FUNCTION_BLOCK PMLStateMachine IMPLEMENTS IPmlStateMachine
VAR_INPUT
END_VAR
VAR_OUTPUT
END_VAR
VAR
	_pmlStateMachine : Tc3_PackML_V2.PML_StateMachine;
	
END_VAR

_pmlStateMachine();

METHOD PUBLIC getState : E_PMLState
VAR_INPUT
END_VAR
getState := _pmlStateMachine.eState;
END_METHOD

METHOD PUBLIC PMLCommand : BOOL
VAR_INPUT
	Command : E_PMLCommand;
END_VAR
_pmlStateMachine.eCommand := Command;
END_METHOD

METHOD PUBLIC StateComplete : BOOL
VAR_INPUT
END_VAR
_pmlStateMachine.M_StateComplete();
END_METHOD

END_FUNCTION_BLOCK

(* stored: Version 1.1.0.1, ProductVersion 3.1.4024.9
   POU PMLStateMachine: Id {52db0bf3-3f38-473f-9975-479dcbeb0e19}, SpecialFunc None
   Method getState: Id {21354818-22a1-4640-b05d-945634b2af00}
   Method PMLCommand: Id {86b656f0-d2a0-4c57-b389-0a32a16cced9}
   Method StateComplete: Id {7a5c1d18-317a-4c03-9289-43fa530749ac} *)
